# EPICS substitutions: streamApp/pluginDb/pluginJPEG.substitutions
#
# pluginJPEG.substitutions
#

file NDFile.template
{
	{
    PORT            = "JPEG\$(N)",
    P               = "$(CAM):",
	R				= "$(PORT):",
    ADDR            = "\$(ADDR=0)",
    TIMEOUT         = "\$(TIMEOUT=1)",
    NDARRAY_PORT    = "\$(PLUGIN_SRC)",
    NDARRAY_ADDR    = "\$(NDARRAY_ADDR=0)",
	}
}
file NDFileAutoFileNumber.template
{
	{
    PORT            = "JPEG\$(N)",
    P               = "$(CAM):",
	R				= "$(PORT):",
	}
}
file NDFileJPEG.template
{
	{
    PORT            = "JPEG\$(N)",
    P               = "$(CAM):",
	R				= "$(PORT):",
    ADDR            = "\$(ADDR=0)",
    TIMEOUT         = "\$(TIMEOUT=1)",
    NDARRAY_PORT    = "\$(PLUGIN_SRC)",
    NDARRAY_ADDR    = "\$(NDARRAY_ADDR=0)",
	}
}
